PROGRAM FuncParoNodoMultidiscos
VAR
	Funci_Multidiscos1:fb_Funciones_Paro;
	Funci_Multidiscos2:fb_Funciones_Paro;
	FunGeneMultidiscos1:FuncGeneralesMultidisc1;
	//Entradas Multidiscos1
	Ftc_Multidiscos1: BOOL;	
	ForzadoFtcMultidiscos1:BOOL;	
	Consenso_Multidiscos1: BOOL;
	//Entradas Multidiscos2
	Ftc2_Multidiscos2: BOOL;
	ForzadoFtc2_Multidiscos2: BOOL;
	Consenso_Multidiscos2: BOOL;
//Entradas Fotocelula libre 1
	Ftc3: BOOL;
	ForzadoFtc3: BOOL;
	Consenso3: BOOL;
//Entradas Fotocelula libre 2
	Ftc4: BOOL;
	ForzadoFtc4: BOOL;
	Consenso4: BOOL;
	
	Multidiscos1StrFuncParoEnviar:StrFuncParoEnviar;
	Multidiscos2StrFuncParoEnviar:StrFuncParoEnviar;
	Libre1StrFuncParoEnviar:StrFuncParoEnviar;
	Libre2StrFuncParoEnviar:StrFuncParoEnviar;	
END_VAR
VAR RETAIN
END_VAR
VAR PERSISTENT 
	HMI_Tiempo_Offset_MParo:INT:=5;
	HMI_TiempoFiltradoFotocel:TIME:=T#2S;
// Generales 
	sModeloActualTabla:STRING;
	sModeloEleccionTabla:STRING;
	sFechaInicModeloTab:STRING;
	sJustificaParoComun:STRING;
END_VAR

//Funciones de paro para cada zona(Fotocelula)

//>>>>>>>>>>>>>>>>>>>>>>>>>>>>>>>>>>>>>>>>>>>>>         	Multidiscos 1         <<<<<<<<<<<<<<<<<<<<<<<<<<<<<<<<<<<<<<<<<<<<<<<<<<<<<<<<<<
Funci_Multidiscos1(Fotocelula:=Ftc_Multidiscos1 OR ForzadoFtcMultidiscos1, 
					Tiempo_Offset_MParo:=HMI_Tiempo_Offset_MParo, 
					TiempoFiltradoFotocel:=HMI_TiempoFiltradoFotocel,
					_StrFuncParoEnviar => Multidiscos1StrFuncParoEnviar,
					S_Justi_Paro_Ftc:=FuncParoNodoCorteH4Remote1.sJustificaParoComun);
					
//>>>>>>>>>>>>>>>>>>>>>>>>>>>>>>>>>>>>>>>>>>>>>         	Multidiscos 2        <<<<<<<<<<<<<<<<<<<<<<<<<<<<<<<<<<<<<<<<<<<<<<<<<<<<<<<<<<
Funci_Multidiscos2(Fotocelula:= Ftc2_Multidiscos2 OR ForzadoFtc2_Multidiscos2,
						Tiempo_Offset_MParo:=HMI_Tiempo_Offset_MParo, 
						TiempoFiltradoFotocel:=HMI_TiempoFiltradoFotocel,
						_StrFuncParoEnviar => Multidiscos2StrFuncParoEnviar,
					S_Justi_Paro_Ftc:=FuncParoNodoMultidiscos.sJustificaParoComun);
						

										
Direccionamiento_variables_com();
Linkado_Entradas();
//FunGeneMultidiscos1(s_JustificaParoComun => sJustificaParoComun,s_ModeloActualTabla => sModeloActualTabla,s_ModeloEleccionTabla => sModeloEleccionTabla);

ACTION Direccionamiento_variables_com:
// Direccionamiento de las variables a la marca que les corresponde donde después se leeran desde el plc maestro



//								>>>>>>>>>>>>>>>>>>>>>>>>>>>>      WORDS    <<<<<<<<<<<<<<<<<<<<<<<<<<<<<<<<

	Var_Com_CH4_MulDis.aWordCom[0]:= INT_TO_WORD (Multidiscos1StrFuncParoEnviar.Cont_Piezas);	    //Contadores de cada fotocelula 
	Var_Com_CH4_MulDis.aWordCom[1]:= INT_TO_WORD (Multidiscos2StrFuncParoEnviar.Cont_Piezas);		//Contadores de cada fotocelula 
	Var_Com_CH4_MulDis.aWordCom[2]:= INT_TO_WORD (Libre1StrFuncParoEnviar.Cont_Piezas);		//Contadores de cada fotocelula 
	Var_Com_CH4_MulDis.aWordCom[3]:= INT_TO_WORD (Libre2StrFuncParoEnviar.Cont_Piezas);		//Contadores de cada fotocelula 
	Var_Com_CH4_MulDis.aWordCom[4]:= INT_TO_WORD (Multidiscos1StrFuncParoEnviar.Min_Parado_Ftc);			//Minutos actuales parado
	Var_Com_CH4_MulDis.aWordCom[5]:= INT_TO_WORD (Multidiscos2StrFuncParoEnviar.Min_Parado_Ftc);			//Minutos actuales parado
	Var_Com_CH4_MulDis.aWordCom[6]:= INT_TO_WORD (Libre1StrFuncParoEnviar.Min_Parado_Ftc);			//Minutos actuales parado
	Var_Com_CH4_MulDis.aWordCom[7]:= INT_TO_WORD (Libre2StrFuncParoEnviar.Min_Parado_Ftc);			//Minutos actuales parado
	
	
	
//                           	>>>>>>>>>>>>>>>>>>>>>>>>>>>>      TIME   <<<<<<<<<<<<<<<<<<<<<<<<<<<<<<<<
	
	
	Var_Com_CH4_MulDis.aTimeCom[0]:=  Multidiscos1StrFuncParoEnviar.t_Entre_Piez_Ftc; 			//Tiempo entre piezas
	Var_Com_CH4_MulDis.aTimeCom[1]:=  Multidiscos2StrFuncParoEnviar.t_Entre_Piez_Ftc;			//Tiempo entre piezas
	Var_Com_CH4_MulDis.aTimeCom[2]:= Libre1StrFuncParoEnviar.t_Entre_Piez_Ftc;				//Tiempo entre piezas
	Var_Com_CH4_MulDis.aTimeCom[3]:= Libre2StrFuncParoEnviar.t_Entre_Piez_Ftc;				//Tiempo entre piezas
	Var_Com_CH4_MulDis.aTimeCom[4]:= Multidiscos1StrFuncParoEnviar.t_Entr_Piez_Ante_Ftc; 		//Tiempo entre piezas anterior
	Var_Com_CH4_MulDis.aTimeCom[5]:= Multidiscos2StrFuncParoEnviar.t_Entr_Piez_Ante_Ftc; 		//Tiempo entre piezas anterior
	Var_Com_CH4_MulDis.aTimeCom[6]:= Libre1StrFuncParoEnviar.t_Entr_Piez_Ante_Ftc; 		//Tiempo entre piezas anterior
	Var_Com_CH4_MulDis.aTimeCom[7]:= Libre2StrFuncParoEnviar.t_Entr_Piez_Ante_Ftc; 		//Tiempo entre piezas anterior
	
	
	
	
//                           	>>>>>>>>>>>>>>>>>>>>>>>>>>>>      STRING  <<<<<<<<<<<<<<<<<<<<<<<<<<<<<<<<
    Var_Com_CH4_MulDis.aStringCom[0] := Multidiscos1StrFuncParoEnviar.H_InParo_Ftc;         //Hora inicio paro 
	Var_Com_CH4_MulDis.aStringCom[1] := Multidiscos2StrFuncParoEnviar.H_InParo_Ftc;         //Hora inicio paro 
	Var_Com_CH4_MulDis.aStringCom[2] := Libre1StrFuncParoEnviar.H_InParo_Ftc;         //Hora inicio paro 
	Var_Com_CH4_MulDis.aStringCom[3] := Libre2StrFuncParoEnviar.H_InParo_Ftc;         //Hora inicio paro 
	Var_Com_CH4_MulDis.aStringCom[4] := Multidiscos1StrFuncParoEnviar.H_FinParo_Ftc;        //Hora Fin paro 
	Var_Com_CH4_MulDis.aStringCom[5] := Multidiscos2StrFuncParoEnviar.H_FinParo_Ftc;        //Hora Fin paro 
	Var_Com_CH4_MulDis.aStringCom[6] := Libre1StrFuncParoEnviar.H_FinParo_Ftc;        //Hora Fin paro 
	Var_Com_CH4_MulDis.aStringCom[7] := Libre2StrFuncParoEnviar.H_FinParo_Ftc;        //Hora Fin paro 
	Var_Com_CH4_MulDis.aStringCom[8] := Multidiscos1StrFuncParoEnviar.S_Justi_Paro_Ftc;		//Justificación del paro
	Var_Com_CH4_MulDis.aStringCom[9] := Multidiscos2StrFuncParoEnviar.S_Justi_Paro_Ftc;		//Justificación del paro
	Var_Com_CH4_MulDis.aStringCom[10] := Libre1StrFuncParoEnviar.S_Justi_Paro_Ftc;		//Justificación del paro
	Var_Com_CH4_MulDis.aStringCom[11] := Libre2StrFuncParoEnviar.S_Justi_Paro_Ftc;		//Justificación del paro
	
	
//                           	>>>>>>>>>>>>>>>>>>>>>>>>>>>>      Bool  <<<<<<<<<<<<<<<<<<<<<<<<<<<<<<<<	

	Var_Com_CH4_MulDis.aBoolCom[0] := Multidiscos1StrFuncParoEnviar.Fotocelula;						//Fotocelula Real
	Var_Com_CH4_MulDis.aBoolCom[1] := Multidiscos2StrFuncParoEnviar.Fotocelula;						//Fotocelula Real
	Var_Com_CH4_MulDis.aBoolCom[2] := Libre1StrFuncParoEnviar.Fotocelula;						//Fotocelula Real
	Var_Com_CH4_MulDis.aBoolCom[3] := Libre2StrFuncParoEnviar.Fotocelula;						//Fotocelula Real
	Var_Com_CH4_MulDis.aBoolCom[4] := Multidiscos1StrFuncParoEnviar.MParo_Ftc;				//Marca de paro 
	Var_Com_CH4_MulDis.aBoolCom[5] := Multidiscos2StrFuncParoEnviar.MParo_Ftc;				//Marca de paro 
	Var_Com_CH4_MulDis.aBoolCom[6] := Libre1StrFuncParoEnviar.MParo_Ftc;				//Marca de paro 
	Var_Com_CH4_MulDis.aBoolCom[7] := Libre2StrFuncParoEnviar.MParo_Ftc;				//Marca de paro 
	Var_Com_CH4_MulDis.aBoolCom[8] := Multidiscos1StrFuncParoEnviar.M_SinParo_Ftc;			//Marca de sin paro activo
	Var_Com_CH4_MulDis.aBoolCom[9] := Multidiscos2StrFuncParoEnviar.M_SinParo_Ftc;			//Marca de sin paro activo
	Var_Com_CH4_MulDis.aBoolCom[10] := Libre1StrFuncParoEnviar.M_SinParo_Ftc;			//Marca de sin paro activo
	Var_Com_CH4_MulDis.aBoolCom[11] := Libre2StrFuncParoEnviar.M_SinParo_Ftc;			//Marca de sin paro activo
	Var_Com_CH4_MulDis.aBoolCom[12] := Multidiscos1StrFuncParoEnviar.tFiltro_up_Ftc;			//Q Temp Up Filtro Fotocelulas
	Var_Com_CH4_MulDis.aBoolCom[13] := Multidiscos2StrFuncParoEnviar.tFiltro_up_Ftc;			//Q Temp Up Filtro Fotocelulas
	Var_Com_CH4_MulDis.aBoolCom[14] := Libre1StrFuncParoEnviar.tFiltro_up_Ftc;			//Q Temp Up Filtro Fotocelulas
	Var_Com_CH4_MulDis.aBoolCom[15] := Libre2StrFuncParoEnviar.tFiltro_up_Ftc;			//Q Temp Up Filtro Fotocelulas
	Var_Com_CH4_MulDis.aBoolCom[16] := Multidiscos1StrFuncParoEnviar.tFiltro_down_Ftc;		//Q Temp Down Filtro Fotocelulas
	Var_Com_CH4_MulDis.aBoolCom[17] := Multidiscos2StrFuncParoEnviar.tFiltro_down_Ftc;		//Q Temp Down Filtro Fotocelulas
	Var_Com_CH4_MulDis.aBoolCom[18] := Libre1StrFuncParoEnviar.tFiltro_down_Ftc;		//Q Temp Down Filtro Fotocelulas
	Var_Com_CH4_MulDis.aBoolCom[19] := Libre2StrFuncParoEnviar.tFiltro_down_Ftc;		//Q Temp Down Filtro Fotocelulas
END_ACTION

ACTION Linkado_Entradas:
// Linkado entradas
Ftc_Multidiscos1:=     MAIN.id0Local.0;
Consenso_Multidiscos1:= TRUE;// main.id0Local2.1;


Ftc2_Multidiscos2:=      MAIN.id0Local.2;
Consenso_Multidiscos2:= TRUE;// main.id0Local2.3;


Ftc3:=      main.id0Local.4;
Consenso3:= TRUE;// main.id0Local2.5;


Ftc4:=      main.id0Local.6;
Consenso4:= TRUE;// main.id0Local2.7;
END_ACTION

END_PROGRAM

(* stored: Version 1.1.0.1, ProductVersion 3.1.4024.12
   POU FuncParoNodoMultidiscos: Id {d0803865-fd7d-4a5f-9349-d5e429b8c6ab}, SpecialFunc None
   Action Direccionamiento_variables_com: Id {ccbcc35e-de58-4535-9514-7aeadbc87591}
   Action Linkado_Entradas: Id {b378cb5d-7ade-49b1-a85b-b3810e171ed5} *)
